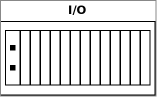
VISUALIZATION VISU_CoverIOSmall  // 157x97
VAR_IN_OUT
	io : CoverIO;
    widget : CoverIOWidget;
END_VAR
    Rectangle (0,21 155x74)
        p3450524324: widget.actualStatus.color.bg
    Rectangle (0,0 155x20), "I/O"
    Rectangle (5,30 15x55), colour variable: widget.coupler.actualStatus.color.bg
    Rectangle (20,30 10x55), colour variable: widget.slot1.actualStatus.color.bg
    Rectangle (30,30 10x55), colour variable: widget.slot2.actualStatus.color.bg
    Rectangle (40,30 10x55), colour variable: widget.slot3.actualStatus.color.bg
    Rectangle (50,30 10x55), colour variable: widget.slot4.actualStatus.color.bg
    Rectangle (60,30 10x55), colour variable: widget.slot5.actualStatus.color.bg
    Rectangle (70,30 10x55), colour variable: widget.slot6.actualStatus.color.bg
    Rectangle (80,30 10x55), colour variable: widget.slot7.actualStatus.color.bg
    Rectangle (90,30 10x55), colour variable: widget.slot8.actualStatus.color.bg
    Rectangle (100,30 10x55), colour variable: widget.slot9.actualStatus.color.bg
    Rectangle (110,30 10x55), colour variable: widget.slot10.actualStatus.color.bg
    Rectangle (120,30 10x55), colour variable: widget.slot11.actualStatus.color.bg
    Rectangle (130,30 10x55), colour variable: widget.slot12.actualStatus.color.bg
    Rectangle (140,30 10x55), colour variable: widget.slot13.actualStatus.color.bg
    Rectangle (10,45 5x5)
    Rectangle (10,65 5x5)
END_VISUALIZATION

(* stored: Version 1.1.0.1, ProductVersion 3.1.0.36
   Visu VISU_CoverIOSmall: Id {b549ff2a-9f66-45e5-bbd1-2826615ebf2c} *)
